FUNCTION F_IEConvert : REAL
VAR_INPUT
	Input																: INT;
	Factor																: REAL;
END_VAR
VAR
END_VAR

// F_IEConvert
// Rev 1.0 - December 28, 2023

F_IEConvert															:= INT_TO_REAL(Input) / Factor;

END_FUNCTION

(* stored: Version 1.1.0.1, ProductVersion 3.1.4024.13
   POU F_IEConvert: Id {1107dc44-afe5-4a12-b5be-d0147952013d}, SpecialFunc None *)
